FUNCTION_BLOCK FB_CenterPosition
VAR_INPUT
	rPositionFront 	: LREAL;
	rPositionBack 	: LREAL;
END_VAR
VAR_OUTPUT
	rPosition 	: LREAL;
	FrontValid 	: BOOL;
	BackValid 	: BOOL;
END_VAR
VAR
	rDistanceBarcodes : LREAL;
END_VAR

FrontValid 	:= TRUE;
BackValid 	:= TRUE;

IF rPositionFront = 0 AND rPosition = 0 THEN
	
	FrontValid 	:= FALSE;
	BackValid 	:= FALSE;
	
	rPosition := -1;
ELSIF rPositionFront = 0 AND rPositionBack <> 0 THEN
	
	FrontValid := FALSE;
	
	rPosition := rPositionBack + (rDistanceBarcodes/2);
ELSIF rPositionFront <> 0 AND rPositionBack = 0 THEN
	
	BackValid := FALSE;
	
	rPosition := rPositionFront - (rDistanceBarcodes/2);
ELSE
	rPosition := (rPositionFront + rPositionBack)/2;
END_IF

END_FUNCTION_BLOCK

(* stored: Version 1.1.0.1
   POU FB_CenterPosition: Id {a8f81790-528b-4d59-93ef-2f6dcb1d7904}, SpecialFunc None *)
